INTERFACE IProcess EXTENDS IObject

{attribute 'monitoring' := 'call'}
{attribute 'OPC.UA.DA.Property' := '1'}
{attribute 'OPC.UA.DA.Access' := '1'}
PROPERTY Busy : BOOL
GET
END_GET
END_PROPERTY

{attribute 'monitoring' := 'call'}
{attribute 'OPC.UA.DA.Property' := '1'}
{attribute 'OPC.UA.DA.Access' := '1'}
PROPERTY Error : BOOL
GET
END_GET
END_PROPERTY

METHOD Execute
END_METHOD

END_INTERFACE

(* stored: Version 1.1.0.1
   Itf IProcess: Id {44e3ce8b-ac1f-4d7c-a60d-08ecae2ae96e}
   Property Busy: Id {51e451a4-81f2-47fb-a17a-20d4804995fb}
   Get Get: Id {8af8039c-c89d-41e0-9d7d-145433c29bed}
   Property Error: Id {ec720c04-807f-445f-ab2a-39f8da91a7e2}
   Get Get: Id {34fec23a-5830-4fef-a20d-8e34142e370a}
   Method Execute: Id {ce1f820d-f7df-4937-80f2-bfbc5db53fec} *)
